PROGRAM MAIN
VAR
	
END_VAR

stackerCraneProcess(
	bHalt:=GVL_ADS.stAdsCom.bHalt,
	bResume:=GVL_ADS.stAdsCom.bResume,
	bStart:=GVL_ADS.stAdsCom.bStart,
	bStop:=GVL_ADS.stAdsCom.bStop,
	fioOutputs:=GVL_IO.fioOutputs,
	fioInputs:=GVL_IO.fioInputs,
	iRackSlot:=GVL_ADS.stAdsCom.iRackSlot,
	iAlgo:=GVL_ADS.stAdsCom.iAlgo,
	iMode:=GVL_ADS.stAdsCom.iMode,
	sCurrentOperation=>GVL_ADS.stAdsCom.sCurrentOperation,
	iPalletsInRack=>GVL_ADS.stAdsCom.iPalletsInRack,
	iTotalPalletsProcessed=>GVL_ADS.stAdsCom.iTotalPalletsProcessed,
	aSlots=>GVL_ADS.stAdsCom.aSlots);

END_PROGRAM

(* stored: Version 1.1.0.1, ProductVersion 3.1.4024.10
   POU MAIN: Id {11a06c43-e2f5-42ce-bb32-02d9d73a9c88}, SpecialFunc None *)
